Staubli VAL3: alarm_action.pgx

program alarm_action()
begin
  stopMove()
  bSuspend=true
  if bPause==true
    bPause=false
  endIf
  read:bCycle=false
  //2015.06.23
  //read:libSave()
  if taskStatus("txtLoad")!=-1
    taskKill("txtLoad")
    wait(taskStatus("txtLoad")==-1)
  endIf
  if taskStatus("motion")!=-1
    taskKill("motion")
    wait(taskStatus("motion")==-1)
  endIf
  call goHome()
end
